// TIA Portal project "KONVEYOR-4" (V17)

(* hardware
DEVICE "HMI_1"  TP700 Comfort
   slot 0: "HMI_1"  TP700 Comfort  6AV2 124-0GC01-0AX0  17.0.0.0
   slot 1: "HMI_RT_1"  TP700 Comfort  6AV2 124-0GC01-0AX0  17.0.0.0
   slot 5: "HMI_1.IE_CP_1"  PROFINET Interface  17.0.0.0
      slot 1: "PROFINET Interface_1"  PROFINET Interface
         slot 1: "Port_1"  Port
         slot 2: "Port_2"  Port
   slot 7: "HMI_1.MPI/DP_CP_1"  MPI/DP Interface  17.0.0.0
DEVICE "S7-1200 station_1"  S7-1200 Station
   slot 0: "Rack_0"  S7-1200 Rack  Rack  V1.0
   slot 1: "PLC_1"  CPU 1214C DC/DC/DC  6ES7 214-1AG40-0XB0  V4.5
*)

// ===== PLC "PLC_1"  CPU 1214C DC/DC/DC =====

VAR_GLOBAL   // PLC tag table "Default tag table"
   "TERMIK" AT %I0.0 : Bool;
   "START/STOP" AT %M20.0 : Bool;
   "ILERI START" AT %M20.1 : Bool;
   "GERI START" AT %M20.2 : Bool;
   "RESET" AT %M20.3 : Bool;
   "MOTOR ILERI" AT %Q0.4 : Bool;
   "MOTOR GERI" AT %Q0.5 : Bool;
   "MOTOR ILERI LAMBA" AT %Q0.0 : Bool;
   "MOTOR GERI LAMBA" AT %Q0.1 : Bool;
   "ARIZA LAMBA" AT %Q0.2 : Bool;
   "ARIZA KORNA" AT %Q0.3 : Bool;
   "ARIZA HAFIZA" AT %M5.0 : Bool;
   "Clock_1Hz" AT %M0.5 : Bool;
   "Tag_1" AT %M90.0 : Bool;
   "DURUMLAMBA" AT %Q0.6 : Bool;
   "Tag_2" AT %M30.1 : Bool;
   "HAREKETSIFIRLA" AT %M30.2 : Bool;
   "Tag_4" AT %M40.1 : Bool;
   "Tag_3" AT %M30.5 : Bool;
END_VAR

DATA_BLOCK "KONVEOR-ANIMASYON"   // DB1
{ S7_Optimized_Access := 'TRUE' }
VERSION : 0.1
   VAR
      "START ILERI" : Bool;
      "HAREKET DEGER" : Int;
      "START GERI" : Bool;
   END_VAR
BEGIN
END_DATA_BLOCK

FUNCTION "KONVEYOR-1" : Void   // FC1, LAD
{ S7_Optimized_Access := 'TRUE' }
VERSION : 0.1
   VAR_INPUT
      TERMIK : Bool;
      STOP : Bool;
      RESET : Bool;
      "ILERI START" : Bool;
      "GERI START" : Bool;
   END_VAR
   VAR_OUTPUT
      "MOTOR ILERI" : Bool;
      "MOTOR ILERI LAMBA" : Bool;
      "MOTOR GERI" : Bool;
      "MOTOR GERI LAMBA" : Bool;
      "ARIZA LAMBA" : Bool;
      "ARIZA KORNA" : Bool;
      DURUMLAMBA : Bool;
   END_VAR
   VAR_TEMP   // added for the SCL form of the ladder/FBD networks
      _w1 : Bool;
   END_VAR
BEGIN

REGION Network 1
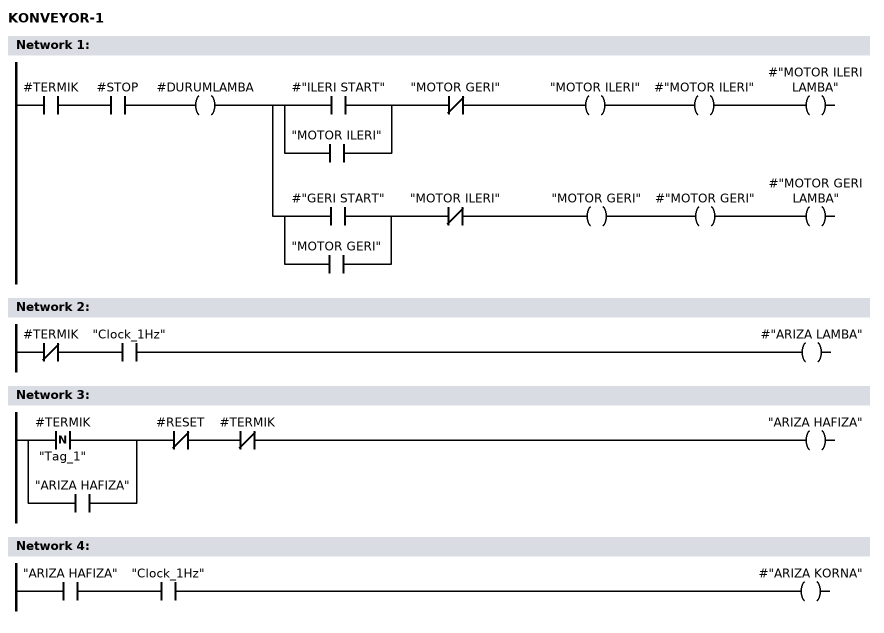
   RUNG wire#powerrail
      Contact( #TERMIK )
      Contact( #STOP )
      Coil( #DURUMLAMBA )
      wire#w1
      Contact( #"ILERI START" )
      wire#w2
      I_Contact( "MOTOR GERI" )
      Coil( "MOTOR ILERI" )
      Coil( #"MOTOR ILERI" )
      Coil( #"MOTOR ILERI LAMBA" )
   END_RUNG
   RUNG wire#w1
      Contact( "MOTOR ILERI" )
   END_RUNG wire#w2
   RUNG wire#w1
      Contact( #"GERI START" )
      wire#w3
      I_Contact( "MOTOR ILERI" )
      Coil( "MOTOR GERI" )
      Coil( #"MOTOR GERI" )
      Coil( #"MOTOR GERI LAMBA" )
   END_RUNG
   RUNG wire#w1
      Contact( "MOTOR GERI" )
   END_RUNG wire#w3
   // the same network as SCL:
   #DURUMLAMBA := #TERMIK AND #STOP;
   "MOTOR ILERI" := #DURUMLAMBA AND (#"ILERI START" OR "MOTOR ILERI") AND NOT "MOTOR GERI";
   #"MOTOR ILERI" := "MOTOR ILERI";
   #"MOTOR ILERI LAMBA" := "MOTOR ILERI";
   "MOTOR GERI" := #DURUMLAMBA AND (#"GERI START" OR "MOTOR GERI") AND NOT "MOTOR ILERI";
   #"MOTOR GERI" := "MOTOR GERI";
   #"MOTOR GERI LAMBA" := "MOTOR GERI";
END_REGION

REGION Network 2
   RUNG wire#powerrail
      I_Contact( #TERMIK )
      Contact( "Clock_1Hz" )
      Coil( #"ARIZA LAMBA" )
   END_RUNG
   // the same network as SCL:
   #"ARIZA LAMBA" := NOT #TERMIK AND "Clock_1Hz";
END_REGION

REGION Network 3
   RUNG wire#powerrail
      N_Contact(operand := #TERMIK, bit := "Tag_1")
      wire#w1
      I_Contact( #RESET )
      I_Contact( #TERMIK )
      Coil( "ARIZA HAFIZA" )
   END_RUNG
   RUNG wire#powerrail
      Contact( "ARIZA HAFIZA" )
   END_RUNG wire#w1
   // the same network as SCL:
   #_w1 := NOT #TERMIK AND "Tag_1";   // falling edge of #TERMIK
   "Tag_1" := #TERMIK;
   "ARIZA HAFIZA" := (#_w1 OR "ARIZA HAFIZA") AND NOT #RESET AND NOT #TERMIK;
END_REGION

REGION Network 4
   RUNG wire#powerrail
      Contact( "ARIZA HAFIZA" )
      Contact( "Clock_1Hz" )
      Coil( #"ARIZA KORNA" )
   END_RUNG
   // the same network as SCL:
   #"ARIZA KORNA" := "ARIZA HAFIZA" AND "Clock_1Hz";
END_REGION
END_FUNCTION

ORGANIZATION_BLOCK "Main"   // OB1, LAD, ProgramCycle
TITLE = "Main Program Sweep (Cycle)"
{ S7_Optimized_Access := 'TRUE' }
VERSION : 0.1
   VAR_INPUT
      Initial_Call : Bool;   // Initial call of this OB
      Remanence : Bool;   // =True, if remanent data are available
   END_VAR
   VAR_TEMP   // added for the SCL form of the ladder/FBD networks
      _w1 : Bool;
   END_VAR
BEGIN

REGION Network 1
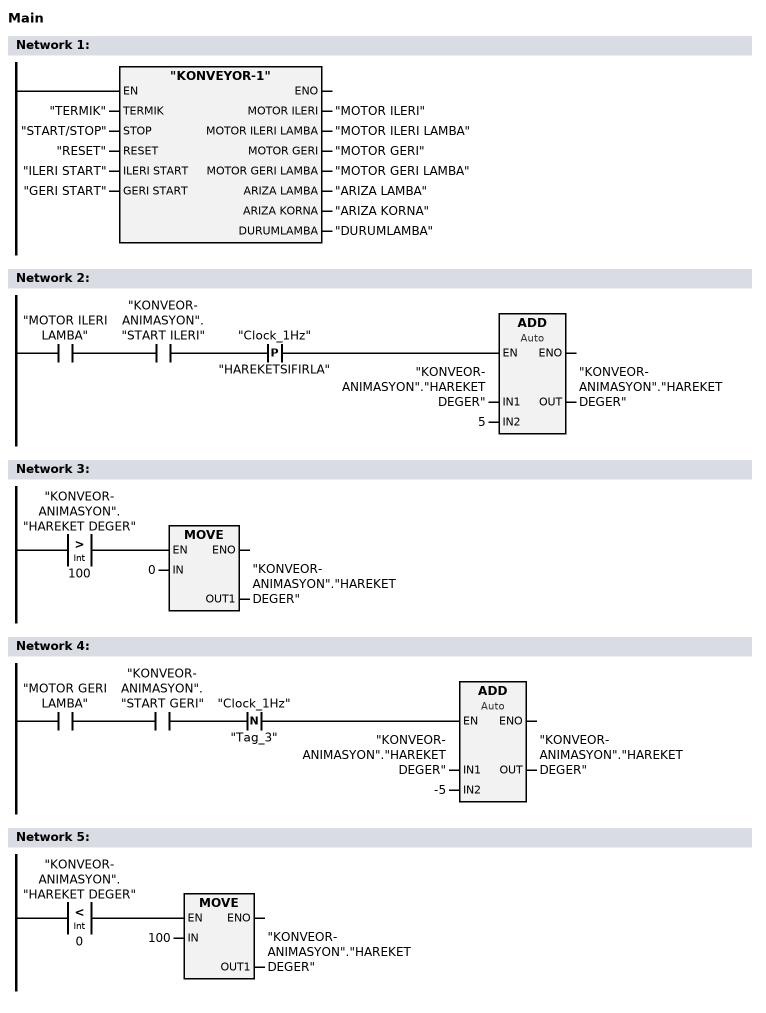
   RUNG wire#powerrail
      "KONVEYOR-1"(TERMIK := "TERMIK", STOP := "START/STOP", RESET := "RESET", "ILERI START" := "ILERI START", "GERI START" := "GERI START", "MOTOR ILERI" => "MOTOR ILERI", "MOTOR ILERI LAMBA" => "MOTOR ILERI LAMBA", "MOTOR GERI" => "MOTOR GERI", "MOTOR GERI LAMBA" => "MOTOR GERI LAMBA", "ARIZA LAMBA" => "ARIZA LAMBA", "ARIZA KORNA" => "ARIZA KORNA", DURUMLAMBA => "DURUMLAMBA")
   END_RUNG
   // the same network as SCL:
   "KONVEYOR-1"(TERMIK := "TERMIK",
                STOP := "START/STOP",
                RESET := "RESET",
                "ILERI START" := "ILERI START",
                "GERI START" := "GERI START",
                "MOTOR ILERI" => "MOTOR ILERI",
                "MOTOR ILERI LAMBA" => "MOTOR ILERI LAMBA",
                "MOTOR GERI" => "MOTOR GERI",
                "MOTOR GERI LAMBA" => "MOTOR GERI LAMBA",
                "ARIZA LAMBA" => "ARIZA LAMBA",
                "ARIZA KORNA" => "ARIZA KORNA",
                DURUMLAMBA => "DURUMLAMBA");
END_REGION

REGION Network 2
   RUNG wire#powerrail
      Contact( "MOTOR ILERI LAMBA" )
      Contact( "KONVEOR-ANIMASYON"."START ILERI" )
      P_Contact(operand := "Clock_1Hz", bit := "HAREKETSIFIRLA")
      Add(in1 := "KONVEOR-ANIMASYON"."HAREKET DEGER", in2 := 5, out => "KONVEOR-ANIMASYON"."HAREKET DEGER")
   END_RUNG
   // the same network as SCL:
   #_w1 := "MOTOR ILERI LAMBA" AND "KONVEOR-ANIMASYON"."START ILERI" AND "Clock_1Hz" AND NOT "HAREKETSIFIRLA";   // rising edge of "Clock_1Hz"
   "HAREKETSIFIRLA" := "Clock_1Hz";
   IF #_w1 THEN "KONVEOR-ANIMASYON"."HAREKET DEGER" := "KONVEOR-ANIMASYON"."HAREKET DEGER" + 5; END_IF;
END_REGION

REGION Network 3
   RUNG wire#powerrail
      { S7_Templates := "SrcType := Int" } GT_Contact(in1 := "KONVEOR-ANIMASYON"."HAREKET DEGER", in2 := 100)
      Move(in := 0, out1 => "KONVEOR-ANIMASYON"."HAREKET DEGER")
   END_RUNG
   // the same network as SCL:
   IF "KONVEOR-ANIMASYON"."HAREKET DEGER" > 100 THEN "KONVEOR-ANIMASYON"."HAREKET DEGER" := 0; END_IF;
END_REGION

REGION Network 4
   RUNG wire#powerrail
      Contact( "MOTOR GERI LAMBA" )
      Contact( "KONVEOR-ANIMASYON"."START GERI" )
      N_Contact(operand := "Clock_1Hz", bit := "Tag_3")
      Add(in1 := "KONVEOR-ANIMASYON"."HAREKET DEGER", in2 := -5, out => "KONVEOR-ANIMASYON"."HAREKET DEGER")
   END_RUNG
   // the same network as SCL:
   #_w1 := "MOTOR GERI LAMBA" AND "KONVEOR-ANIMASYON"."START GERI" AND NOT "Clock_1Hz" AND "Tag_3";   // falling edge of "Clock_1Hz"
   "Tag_3" := "Clock_1Hz";
   IF #_w1 THEN "KONVEOR-ANIMASYON"."HAREKET DEGER" := "KONVEOR-ANIMASYON"."HAREKET DEGER" + (-5); END_IF;
END_REGION

REGION Network 5
   RUNG wire#powerrail
      { S7_Templates := "SrcType := Int" } LT_Contact(in1 := "KONVEOR-ANIMASYON"."HAREKET DEGER", in2 := 0)
      Move(in := 100, out1 => "KONVEOR-ANIMASYON"."HAREKET DEGER")
   END_RUNG
   // the same network as SCL:
   IF "KONVEOR-ANIMASYON"."HAREKET DEGER" < 0 THEN "KONVEOR-ANIMASYON"."HAREKET DEGER" := 100; END_IF;
END_REGION
END_ORGANIZATION_BLOCK

(* ===== HMI "HMI_RT_1" =====
system functions are stored by id; their names below are inferred from use
connection "HMI_Connection_1": ETHERNET, S7_1200_OMS

HMI tags "Default tag table"
   "Tag_ScreenNumber" : UInt, internal
   "START/STOP" : Bool = PLC "START/STOP" AT %M20.0, 100 ms
   "ILERI START" : Bool = PLC "ILERI START" AT %M20.1, 1 s
   "GERI START" : Bool = PLC "GERI START" AT %M20.2, 1 s
   "RESET" : Bool = PLC RESET AT %M20.3, 1 s
   "MOTOR ILERI" : Bool = PLC "MOTOR ILERI" AT %Q0.4, 1 s
   "MOTOR GERI" : Bool = PLC "MOTOR GERI" AT %Q0.5, 1 s
   "buttonisim" : UInt, internal
   "ARIZA LAMBA" : Bool = PLC "ARIZA LAMBA" AT %Q0.2, 100 ms
   "ARIZA KORNA" : Bool = PLC "ARIZA KORNA" AT %Q0.3, 100 ms
   "TERMIK" : Bool = PLC TERMIK AT %I0.0, 100 ms
   "DURUMLAMBA" : Bool = PLC DURUMLAMBA AT %Q0.6, 100 ms
   "MOTOR ILERI LAMBA" : Bool = PLC "MOTOR ILERI LAMBA" AT %Q0.0, 1 s
   "KONVEOR-ANIMASYON_HAREKET DEGER" : Int = PLC "KONVEOR-ANIMASYON"."HAREKET DEGER", 100 ms
   "KONVEOR-ANIMASYON_START" : Bool = PLC "KONVEOR-ANIMASYON"."START ILERI", 100 ms
   "KONVEOR-ANIMASYON_START GERI" : Bool = PLC "KONVEOR-ANIMASYON"."START GERI", 1 s

screen "Root screen" 800x420, template "Template_1"
   on GenerateScreen: SetTag("Tag_ScreenNumber", 1)
   Button "Button_4" at 608,292 size 137x44; TextOff 'RESET'
      on Press: SetBit("RESET")
      on Release: ResetBit("RESET")
   TextField "Text field_4" at 138,8 size 524x40; Text 'KONVEYÖR KONTROL'
   GraphicView "Graphic view_2" at 23,239 size 518x50; Picture "Graphic_1"
      Appearance <- "MOTOR ILERI LAMBA"
   Rectangle "Rectangle_1" at 106,209 size 55x46
      HorizontalMovement <- "KONVEOR-ANIMASYON_HAREKET DEGER"
   Button "Button_5" at 32,61 size 137x44; TextOn 'DURUDUR'; TextOff 'ON / OFF'; TextList "Text_list_2"
      ProcessValue <- "buttonisim"
      on Click: InvertBit("START/STOP"); ResetBit("KONVEOR-ANIMASYON_START"); ResetBit("KONVEOR-ANIMASYON_START GERI")
   GraphicIOField "PlotLight_Round_G_3" at 76,116 size 50x50; PictureOff "PilotLight_Round_R_On_256c"; PictureOn "PilotLight_Round_G_On_256c"
      ProcessValue <- "DURUMLAMBA"
   Button "Button_2" at 213,61 size 137x44; TextOff 'ILERI'
      on Press: SetBit("ILERI START"); SetBit("KONVEOR-ANIMASYON_START")
      on Release: ResetBit("ILERI START")
   GraphicIOField "PlotLight_Round_G_1" at 258,119 size 50x50; PictureOn "PilotLight_Round_G_On_256c"; PictureOff "PilotLight_Round_R_On_256c"
      ProcessValue <- "MOTOR ILERI"
   Button "Button_3" at 395,61 size 137x44; TextOff 'GERI'
      on Press: SetBit("GERI START"); SetBit("KONVEOR-ANIMASYON_START GERI")
      on Release: ResetBit("GERI START")
   GraphicIOField "PlotLight_Round_G_4" at 439,116 size 50x50; PictureOn "PilotLight_Round_G_On_256c"; PictureOff "PilotLight_Round_R_On_256c"
      ProcessValue <- "MOTOR GERI"
   GraphicIOField "PlotLight_Round_R_2" at 727,58 size 50x50; PictureOff "PilotLight_Round_R_On_256c"
      ProcessValue <- "TERMIK"
   GraphicIOField "PlotLight_Round_R" at 727,206 size 50x50; PictureOn "PilotLight_Round_R_On_256c"
      ProcessValue <- "ARIZA KORNA"
   TextField "Text field_2" at 575,217 size 143x27; Text 'KORNA'
   TextField "Text field_1" at 575,143 size 148x27; Text 'ARIZA'
   TextField "Text field_3" at 575,69 size 165x27; Text 'TERMİK'
   GraphicIOField "PlotLight_Round_R_4" at 727,132 size 50x50; PictureOn "PilotLight_Round_R_On_256c"
      ProcessValue <- "ARIZA LAMBA"

Template "Template_1" 800x420
   Button "Exit" at 720,360 size 78x58; TextOff 'Exit'; PictureOff "ExitRuntime_TP700_Comfort_TR"; PictureOn "ExitRuntime_TP700_Comfort_TR"
      on Release: StopRuntime(0)
   Button "Template_Button" at 640,360 size 78x58; TextOff 'Text'
   Button "Template_Button_1" at 560,360 size 78x58; TextOff 'Text'
   Button "Template_Button_2" at 480,360 size 78x58; TextOff 'Text'
   Button "Template_Button_3" at 400,360 size 78x58; TextOff 'Text'
   Button "Template_Button_4" at 321,360 size 78x58; TextOff 'Text'
   Button "Template_Button_5" at 241,360 size 78x58; TextOff 'Text'
   Button "Template_Button_6" at 161,360 size 78x58; TextOff 'Text'
   Button "Alarms" at 81,360 size 78x58; TextOff 'Alarms'; PictureOff "AlarmDisplay_TP700_Comfort_TR"; PictureOn "AlarmDisplay_TP700_Comfort_TR"
      on Release: function_ef3f5d25("Alarm window_Unacknowledged", -1)
   Button "Start screen" at 1,360 size 78x58; TextOff 'Start screen'; PictureOff "NavigateHome_TP700_Comfort_TR"; PictureOn "NavigateHome_TP700_Comfort_TR"
      on Release: ActivateScreen("Root screen", 0)
*)